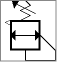
VISUALIZATION VISU_M1Figure_Regulator  // 57x62
    Rectangle (10,20 30x30)
    Line (15,35) (35,35)
    Line (25,50) (25,60)
    Line (25,60) (55,60)
    Line (55,50) (55,60)
    Line (55,50) (40,35)
    Line (20,20) (30,15)
    Line (20,10) (30,15)
    Line (20,10) (30,5)
    Line (25,0) (30,5)
    Line (15,3) (35,13)
    Polygon (14,8) (12,1) (19,0)
    Polygon (10,25) (5,22) (10,20)
    Polygon (15,40) (10,35) (15,30)
    Polygon (35,40) (40,35) (35,30)
END_VISUALIZATION

(* stored: Version 1.1.0.1, ProductVersion 3.1.4019.2
   Visu VISU_M1Figure_Regulator: Id {b4051ab5-03e9-4174-8068-0077f5457036} *)
